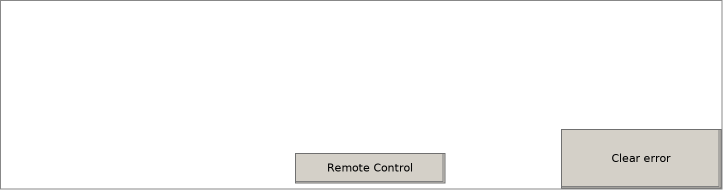
VISUALIZATION Visualization  // 723x190
    Button (295,153 150x30), "Remote Control"
        toggle bRemote
    Button (561,129 160x59), "Clear error"
END_VISUALIZATION

(* stored: Version 1.1.0.1, ProductVersion 3.1.4022.18
   Visu Visualization: Id {efb5648a-2a78-4c47-92e0-aefd85daf6f2} *)
